// TIA Portal V20 export
// export: Created 2025-12-01T14:56:22.0331015Z, ExportSetting None, DisplayName Totally Integrated Automation Portal, DisplayVersion V20 Update 3, DisplayName TIA Portal Openness, DisplayVersion V20 Update 3, DisplayName TIA Portal Version Control Interface, DisplayVersion V20 Update 3, DisplayName STEP 7 Professional, DisplayVersion V20 Update 3, DisplayName STEP 7 Safety, DisplayVersion V20 Update 2, DisplayName WinCC Basic/Comfort/Advanced, DisplayVersion V20 Update 3, DisplayName WinCC Professional, DisplayVersion V20 Update 3, DisplayName WinCC Unified, DisplayVersion V20 Update 3
TYPE "NDD_Enfardadora_Output"
   STRUCT
      BitDeVida : Bool;
      Libre_01 : Bool;
      Libre_02 : Bool;
      Libre_03 : Bool;
      Libre_04 : Bool;
      Libre_05 : Bool;
      Libre_06 : Bool;
      Libre_07 : Bool;
      AutomaticoSinAnomalisas : Bool;
      EnAutomico : Bool;   // Libre_11
      ElevadorEnMovimiento : Bool;
      PaletaPosicionEnvolver : Bool;
      DescendiendoElevador : Bool;
      RealizandoCapa : Bool;
      AscendiendoElevador : Bool;
      Libre_17 : Bool;
      PaletaEvacuada : Bool;
      StopEnfardadora : Bool;
      MarchaEnfardadora : Bool;
      Check_EnEnfardadora : Bool;
      "FinEnfardado(Rearme)" : Bool;
      "EmpezarEnfardado(Rearme)" : Bool;
      "ContiuarEnfardado(Rearme)" : Bool;
      IrPosicionHome : Bool;
      Libre_30 : Bool;
      Libre_31 : Bool;
      Libre_32 : Bool;
      Libre_33 : Bool;
      Libre_34 : Bool;
      Libre_35 : Bool;
      Libre_36 : Bool;
      Libre_37 : Bool;
      AlturaPaleta : Int;
      AlturaElevador : Int;
      Programa : Int;
   END_STRUCT;
END_TYPE
